FUNCTION_BLOCK TaskFB EXTENDS TaskBase 
VAR_INPUT
END_VAR
VAR_OUTPUT
END_VAR
VAR
END_VAR

END_FUNCTION_BLOCK

(* stored: Version 1.1.0.1, ProductVersion 3.1.4024.12
   POU TaskFB: Id {6462aa7d-109a-4387-98ec-58b721f7df0e}, SpecialFunc None *)
